FUNCTION F_SAFETY_StatusFB_TO_ESTOP : ST_SAFETY_FBESTOP 	(* Struktura dedykowana *)
VAR_INPUT
	stFBStatus						: ST_SAFETY_FBStatus; 	(* Struktura ogolna *)
END_VAR

F_SAFETY_StatusFB_TO_ESTOP.uStatus.stStatusWords	:= stFBStatus;									(* Przepisanie *)
F_SAFETY_StatusFB_TO_ESTOP.eState 					:= stFBStatus.BState;							(* Ustawienie enum *)
F_SAFETY_StatusFB_TO_ESTOP.bGeneralError			:= stFBStatus.wDiagnosis <> 0;					(* General Error *)

END_FUNCTION

(* stored: Version 1.1.0.1, ProductVersion 3.1.4022.12
   POU F_SAFETY_StatusFB_TO_ESTOP: Id {a038978e-c779-4940-950d-642f86327372}, SpecialFunc None *)
